(* Logix 5000 project; controller ARS14002_PLC vendor 1 type 14 code 218 rev 30.11; software revision 30.01; part 3 of 13 *)
(* tags used below, declared in another part *)
   AC_OK_1000 : BOOL;
   AC_OK_600 : BOOL;
   AC_OK_800 : BOOL;
   AC_OK_MCP : BOOL;
   AN_1000A : CM_AI_SCL;
   AN_1000B : CM_AI_SCL;
   AN_1000C : CM_AI_SCL;
   AN_101A : CM_AI_SCL;
   AN_101B : CM_AI_SCL;
   AN_101C : CM_AI_SCL;
   AN_200A : CM_AI_SCL;
   ARS_TO_AT3 : UDT_IPC;
   AT2_ATOMIZE_FLOW : REAL;
   AT2_ATOMIZE_FLOW_SCFM : REAL;
   AT2_CHAMBER_PRESSURE : REAL;
   AT2_COMM_STATUS_CONS : BOOL;
   AT2_COMM_STATUS_PROD : BOOL;
   AT2_END_ATOMIZATION : BOOL;
   AT2_HIBON_DISCHARGE_TEMP : REAL;
   AT2_HIBON_INSERTION_VALVE_OPEN : BOOL;
   AT2_HIBON_RUNNING : BOOL;
   AT2_INLET_FLOW : REAL;
   AT2_INLET_FLOW_SCFM : REAL;
   AT2_INLET_VALVE_OPEN : BOOL;
   AT2_PARTICULATE_POST_CYCLONE : REAL;
   AT2_PARTICULATE_POST_FILTER : REAL;
   AT2_PEDESTAL_LEVEL : REAL;
   AT2_PRAXAIR_PRESSURE : REAL;
   AT2_PRESTART : BOOL;
   AT2_START_ATOMIZATION : BOOL;
   AT2_V1_OPEN : BOOL;
   AT2_V4_OPEN : BOOL;
   AT3_ATOMIZE_FLOW : REAL;
   AT3_ATOMIZE_FLOW_SCFM : REAL;
   AT3_ATOMIZE_VALVE_OPEN : BOOL;
   AT3_CHAMBER_PRESSURE : REAL;
   AT3_CHAMBER_VACUUM : REAL;
   AT3_COMM_STATUS_CONS : BOOL;
   AT3_COMM_STATUS_PROD : BOOL;
   AT3_END_ATOMIZATION : BOOL;
   AT3_HIBON_DISCHARGE_TEMP : REAL;
   AT3_HIBON_INSERTION_VALVE_OPEN : BOOL;
   AT3_HIBON_RUNNING : BOOL;
   AT3_INLET_FLOW : REAL;
   AT3_INLET_FLOW_SCFM : REAL;
   AT3_INLET_VALVE_OPEN : BOOL;
   AT3_MELT_STATUS : BOOL;
   AT3_PARTICULATE_POST_CYCLONE : REAL;
   AT3_PARTICULATE_POST_FILTER : REAL;
   AT3_PEDESTAL_LEVEL : REAL;
   AT3_PRESTART : BOOL;
   AT3_START_ATOMIZATION : BOOL;
   AT3_TO_ARS : UDT_IPC;
   AT3_V1_OPEN : BOOL;
   AT3_V4_OPEN : BOOL;
   DC_OK_1000 : BOOL;
   DC_OK_600 : BOOL;
   DC_OK_800 : BOOL;
   DC_OK_MCP : BOOL;
   Deoxo_CurrentState : DINT;
   Deoxo_TransitionState : DINT;
   ESTOP_1 : BOOL;   // Pump Skid E-Stops
   ESTOP_2 : BOOL;   // FAN/HXR E-Stops
   ew_test_200 : BOOL;
   FSL_1000B : BOOL;
   FT_1002 : CM_AI_SCL;
   FT_1221 : CM_AI_SCL;
   FT_1251 : CM_AI_SCL;
   FT_202 : CM_AI_SCL;
   FT_202_ALT_SCFM : REAL;
   FT_502 : CM_AI_SCL;
   FT_502_ALT_SCFM : REAL;
   FT_904 : CM_AI_SCL;
   HXR_1250 : CM_DO_FVNR;
   IT_1250 : CM_AI_SCL;
   MTR_550 : CM_DO_FVNR;
   P_800A_RUN_OCCURRED : BOOL;
   P_800B_RUN_OCCURRED : BOOL;
   P_800C : CM_DO_FVR;
   P_800C_RUN_OCCURRED : BOOL;
   P_800D : CM_DO_FVR;
   P_800D_RUN_OCCURRED : BOOL;
   PDT_1101A : CM_AI_SCL_ALT;
   PDT_1301A : CM_AI_SCL_ALT;
   PDT_1301B : CM_AI_SCL_ALT;
   PDT_601 : CM_AI_SCL_ALT;
   PDT_603 : CM_AI_SCL_ALT;
   PDT_603_PERCENT : REAL;
   PDT_701 : CM_AI_SCL_ALT;
   PDT_701_ALT_GAL : REAL;
   PDT_701_ALT_SCF : REAL;
   PDT_721_CALC : REAL;
   PDT_751 : CM_AI_SCL_ALT;
   PDT_753 : CM_AI_SCL_ALT;
   PILOT_ATOMIZE_VALVE_OPEN : BOOL;   // Halo Valve
   PILOT_COMM_STATUS : BOOL;
   PILOT_EXHAUST_VALVE_OPEN : BOOL;
   PILOT_INLET_VALVE_OPEN : BOOL;   // Pressure Control Status (Backfill)
   PILOT_PARTICULATE_POST_FILTER : REAL;
   PILOT_PEDESTAL_LEVEL : REAL;
   PT_051 : CM_AI_SCL;
   PT_1001 : CM_AI_SCL;
   PT_1002 : CM_AI_SCL;
   PT_1003 : CM_AI_SCL;
   PT_101A : CM_AI_SCL;
   PT_101B : CM_AI_SCL;
   PT_101C : CM_AI_SCL;
   PT_1101A : CM_AI_SCL;
   PT_1201 : CM_AI_SCL;
   PT_1220 : CM_AI_SCL;
   PT_1222 : CM_AI_SCL;
   PT_1301A : CM_AI_SCL;
   PT_1301B : CM_AI_SCL;
   PT_201 : CM_AI_SCL;
   PT_222 : CM_AI_SCL;
   PT_601 : CM_AI_SCL;
   PT_601_LR : CM_AI_SCL;
   PT_603 : CM_AI_SCL;
   PT_701 : CM_AI_SCL;
   PT_721 : CM_AI_SCL;
   PT_751 : CM_AI_SCL;
   PT_753 : CM_AI_SCL;
   PT_802A : CM_AI_SCL;
   PT_802B : CM_AI_SCL;
   PT_802C : CM_AI_SCL;
   PT_802D : CM_AI_SCL;
   PT_803 : CM_AI_SCL;
   PT_806 : CM_AI_SCL;
   PT_902 : CM_AI_SCL;
   SCR_1250 : BOOL;   // HXR-1250 SCR Active Signal
   TE_1003 : CM_AI_SCL;
   TE_101A : CM_AI_SCL;
   TE_101B : CM_AI_SCL;
   TE_101C : CM_AI_SCL;
   TE_1201 : CM_AI_SCL;
   TE_1202 : CM_AI_SCL;
   TE_1203 : CM_AI_SCL;
   TE_1204 : CM_AI_SCL;
   TE_1205 : CM_AI_SCL;
   TE_1206 : CM_AI_SCL;
   TE_1250A : CM_AI_SCL;
   TE_1250B : CM_AI_SCL;
   TE_1252 : CM_AI_SCL;
   TE_501 : CM_AI_SCL;
   TE_504 : CM_AI_SCL;
   TE_601 : CM_AI_SCL;
   TE_602 : CM_AI_SCL;
   TE_604 : CM_AI_SCL;
   TE_609 : CM_AI_SCL;
   TE_801A : CM_AI_SCL;
   TE_801B : CM_AI_SCL;
   TE_801C : CM_AI_SCL;
   TE_801D : CM_AI_SCL;
   TE_802A : CM_AI_SCL;
   TE_802B : CM_AI_SCL;
   TE_802C : CM_AI_SCL;
   TE_802D : CM_AI_SCL;
   TE_803A : CM_AI_SCL;
   TE_803B : CM_AI_SCL;
   TE_803C : CM_AI_SCL;
   TE_803D : CM_AI_SCL;
   TE_804A : CM_AI_SCL;
   TE_804B : CM_AI_SCL;
   TE_804C : CM_AI_SCL;
   TE_804D : CM_AI_SCL;
   TE_901 : CM_AI_SCL;
   TE_902 : CM_AI_SCL;
   TE_903 : CM_AI_SCL;
   TE_904 : CM_AI_SCL;
   TE_T_RAWMAX : INT;
   TE_T_RAWMIN : INT;
   TK_1000_SCF : REAL;   // TOTAL SCF IN BUFFER
   VAPORIZER_WATER_DIFFERENTIAL : REAL;
   WATCHDOG_IN_100 : BOOL;
   WATCHDOG_IN_1000 : BOOL;
   WATCHDOG_IN_600 : BOOL;
   WATCHDOG_IN_800 : BOOL;
   XV_1001 : CM_DO_VLV;
   XV_101B : CM_DO_VLV;
   XV_101C : CM_DO_VLV;
   XV_1123 : CM_DO_VLV;
   XV_1201 : CM_DO_VLV;
   XV_1202 : CM_DO_VLV;
   XV_1203 : CM_DO_VLV;
   XV_1204 : CM_DO_VLV;
   XV_1205 : CM_DO_VLV;
   XV_623 : CM_DO_VLV;
   XV_703 : CM_DO_VLV;
   XV_721A : CM_DO_VLV;
   XV_721B : CM_DO_VLV;
   XV_801A : CM_DO_VLV;
   XV_801B : CM_DO_VLV;
   XV_801C : CM_DO_VLV;
   XV_801D : CM_DO_VLV;
   XV_806 : CM_DO_VLV;
   ZT_1001 : CM_AI_SCL;
   ZT_1002 : CM_AI_SCL;
   ZT_101A : CM_AI_SCL;
   ZT_101B : CM_AI_SCL;
   ZT_101C : CM_AI_SCL;
   ZT_102A : CM_AI_SCL;
   ZT_102B : CM_AI_SCL;
   ZT_102C : CM_AI_SCL;
   ZT_1221 : CM_AI_SCL;
   ZT_1251 : CM_AI_SCL;
   ZT_202 : CM_AI_SCL;
   ZT_204 : CM_AI_SCL;
   ZT_207 : CM_AI_SCL;
   ZT_504 : CM_AI_SCL;
   ZT_603 : CM_AI_SCL;
   ZT_605 : CM_AI_SCL;
   ZT_753 : CM_AI_SCL;
   ZT_754 : CM_AI_SCL;
   ZT_755 : CM_AI_SCL;
(* MainProgPeriodic, continued *)

ROUTINE MainRoutinePeriodic   (* ladder *)
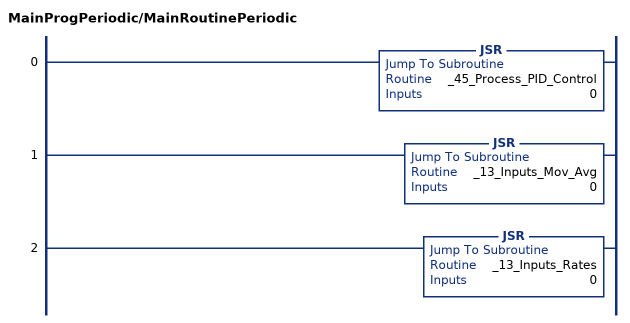
   0: JSR(_45_Process_PID_Control,0);
   1: JSR(_13_Inputs_Mov_Avg,0);
   2: JSR(_13_Inputs_Rates,0);
END_ROUTINE
END_PROGRAM

PROGRAM MainProgram   (* main routine MainRoutine *)
VAR
   BAND_01 : FBD_BOOLEAN_AND := (In3 := 1, In4 := 1, In5 := 1, In6 := 1, In7 := 1, In8 := 1);
   BNOT_01 : FBD_BOOLEAN_NOT := (Out := 1);
   BNOT_02 : FBD_BOOLEAN_NOT := (Out := 1);
   BNOT_03 : FBD_BOOLEAN_NOT := (Out := 1);
   BNOT_04 : FBD_BOOLEAN_NOT := (Out := 1);
   BOR_01 : FBD_BOOLEAN_OR;
   BOR_02 : FBD_BOOLEAN_OR;
   delete_ARS_DERIME_AUTO : BOOL;
   delete_AT2_PLANT_MAX_H2O : REAL := -85.0;
   delete_AT2_PLANT_MAX_O2 : REAL;
   delete_AT3_PLANT_MAX_H2O : REAL := -85.0;
   delete_AT3_PLANT_MAX_O2 : REAL;
   delete_PILOT_PLANT_MAX_H2O : REAL := -85.0;
   delete_PILOT_PLANT_MAX_O2 : REAL;
   delete_XV_623_FILL_MODE : BOOL;   // 0 = VENT 1 = FILL
   DERIME_EMPTY : BOOL;
   DERIME_EMPTY_ALARM : BOOL;
   DERIME_EMPTY_HOLD_TMR : TIMER := (PRE := 300000);
   DERIME_FILL : BOOL;
   DERIME_FULL : BOOL;
   DERIME_FULL_ALARM : BOOL;
   DERIME_FULL_HOLD_TMR : TIMER := (PRE := 600000);
   DERIME_SPH : REAL := 40.0;
   DERIME_SPL : REAL := 5.0;
   DERIME_VENT : BOOL := 1;
   DERV_01 : DERIVATIVE := (Gain := 1.0, RTSTime := 1);
   MAVE_01 : MOVING_AVERAGE := (SampleEnable := 1, NumberOfSamples := 1);
   MAVE_02 : MOVING_AVERAGE := (SampleEnable := 1, NumberOfSamples := 1);
   PT_701_DERIME_VENT_SPH : REAL := 30.0;
   PT_701_DERIME_VENT_SPL : REAL := 5.0;
   XV_721_BURP_TMR : TIMER;
END_VAR

ROUTINE _00_Startup   (* ladder *)
// Initialization Routines
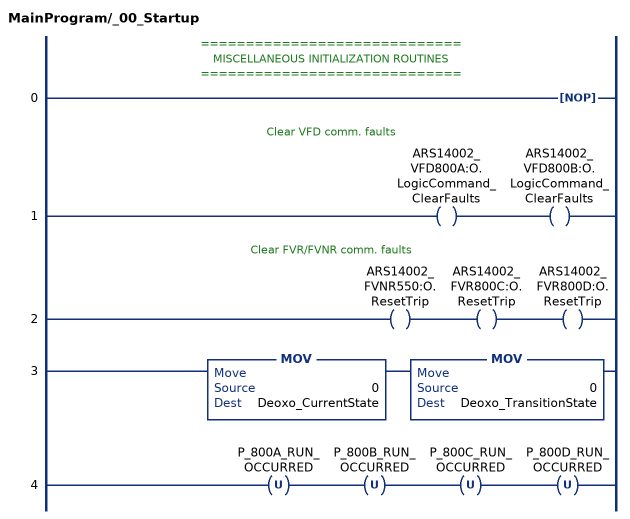
   // =============================
   // MISCELLANEOUS INITIALIZATION ROUTINES
   // =============================
   0: NOP();
   // Clear VFD comm. faults
   1: OTE(ARS14002_VFD800A:O.LogicCommand_ClearFaults)OTE(ARS14002_VFD800B:O.LogicCommand_ClearFaults);
   // Clear FVR/FVNR comm. faults
   2: OTE(ARS14002_FVNR550:O.ResetTrip)OTE(ARS14002_FVR800C:O.ResetTrip)OTE(ARS14002_FVR800D:O.ResetTrip);
   3: MOV(0,Deoxo_CurrentState)MOV(0,Deoxo_TransitionState);
   4: OTU(P_800A_RUN_OCCURRED)OTU(P_800B_RUN_OCCURRED)OTU(P_800C_RUN_OCCURRED)OTU(P_800D_RUN_OCCURRED);
END_ROUTINE

ROUTINE _10_Inputs_Analog   (* ladder *)
// Analog Input scaling and alarm handling routine
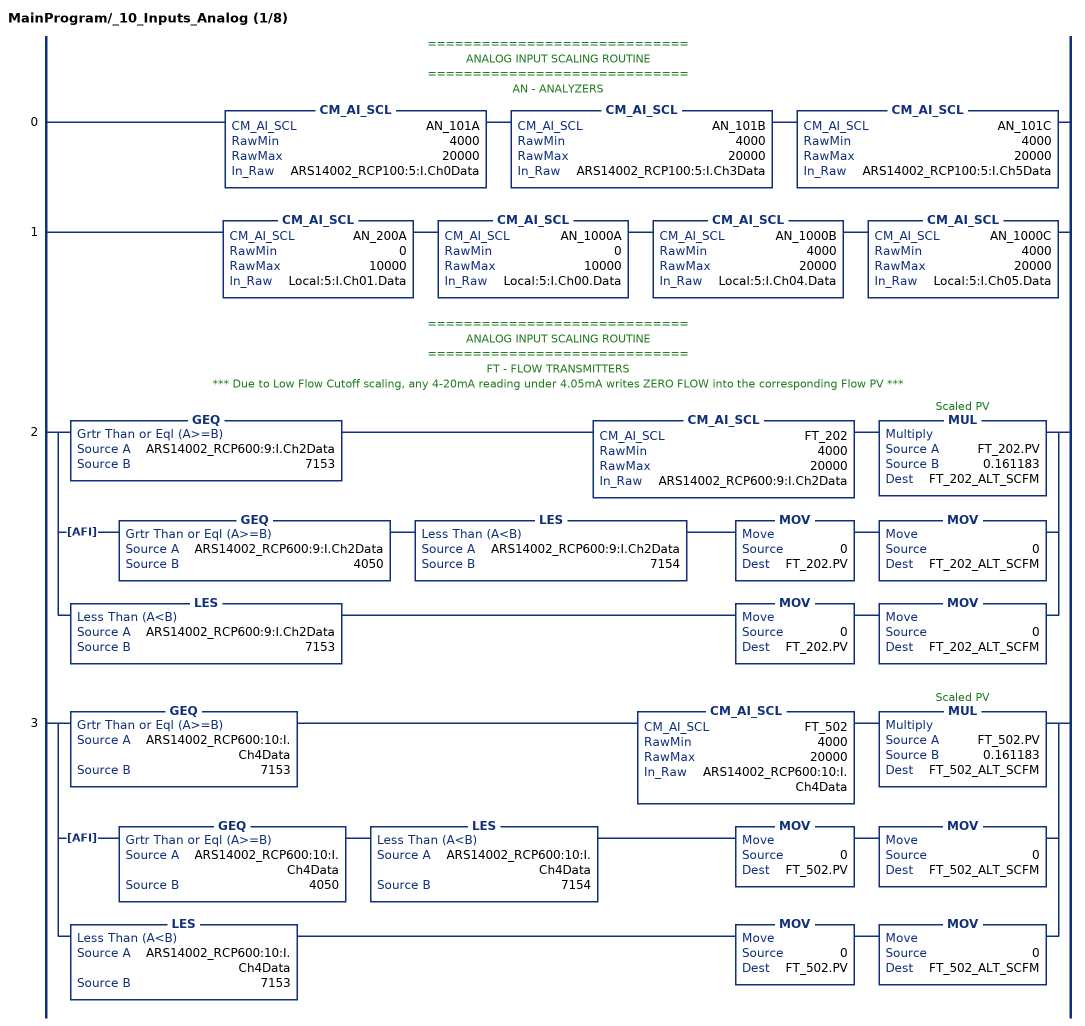
   // =============================
   // ANALOG INPUT SCALING ROUTINE
   // =============================
   // AN - ANALYZERS
   0: CM_AI_SCL(AN_101A,4000,20000,ARS14002_RCP100:5:I.Ch0Data)CM_AI_SCL(AN_101B,4000,20000,ARS14002_RCP100:5:I.Ch3Data)CM_AI_SCL(AN_101C,4000,20000,ARS14002_RCP100:5:I.Ch5Data);
   1: CM_AI_SCL(AN_200A,0,10000,Local:5:I.Ch01.Data)CM_AI_SCL(AN_1000A,0,10000,Local:5:I.Ch00.Data)CM_AI_SCL(AN_1000B,4000,20000,Local:5:I.Ch04.Data)CM_AI_SCL(AN_1000C,4000,20000,Local:5:I.Ch05.Data);
   // =============================
   // ANALOG INPUT SCALING ROUTINE
   // =============================
   // FT - FLOW TRANSMITTERS
   // *** Due to Low Flow Cutoff scaling, any 4-20mA reading under 4.05mA writes ZERO FLOW into the corresponding Flow PV ***
   2: [GEQ(ARS14002_RCP600:9:I.Ch2Data,7153) CM_AI_SCL(FT_202,4000,20000,ARS14002_RCP600:9:I.Ch2Data) MUL(FT_202.PV,0.161183,FT_202_ALT_SCFM) ,AFI() GEQ(ARS14002_RCP600:9:I.Ch2Data,4050) LES(ARS14002_RCP600:9:I.Ch2Data,7154) MOV(0,FT_202.PV) MOV(0,FT_202_ALT_SCFM) ,LES(ARS14002_RCP600:9:I.Ch2Data,7153) MOV(0,FT_202.PV) MOV(0,FT_202_ALT_SCFM) ];
   3: [GEQ(ARS14002_RCP600:10:I.Ch4Data,7153) CM_AI_SCL(FT_502,4000,20000,ARS14002_RCP600:10:I.Ch4Data) MUL(FT_502.PV,0.161183,FT_502_ALT_SCFM) ,AFI() GEQ(ARS14002_RCP600:10:I.Ch4Data,4050) LES(ARS14002_RCP600:10:I.Ch4Data,7154) MOV(0,FT_502.PV) MOV(0,FT_502_ALT_SCFM) ,LES(ARS14002_RCP600:10:I.Ch4Data,7153) MOV(0,FT_502.PV) MOV(0,FT_502_ALT_SCFM) ];
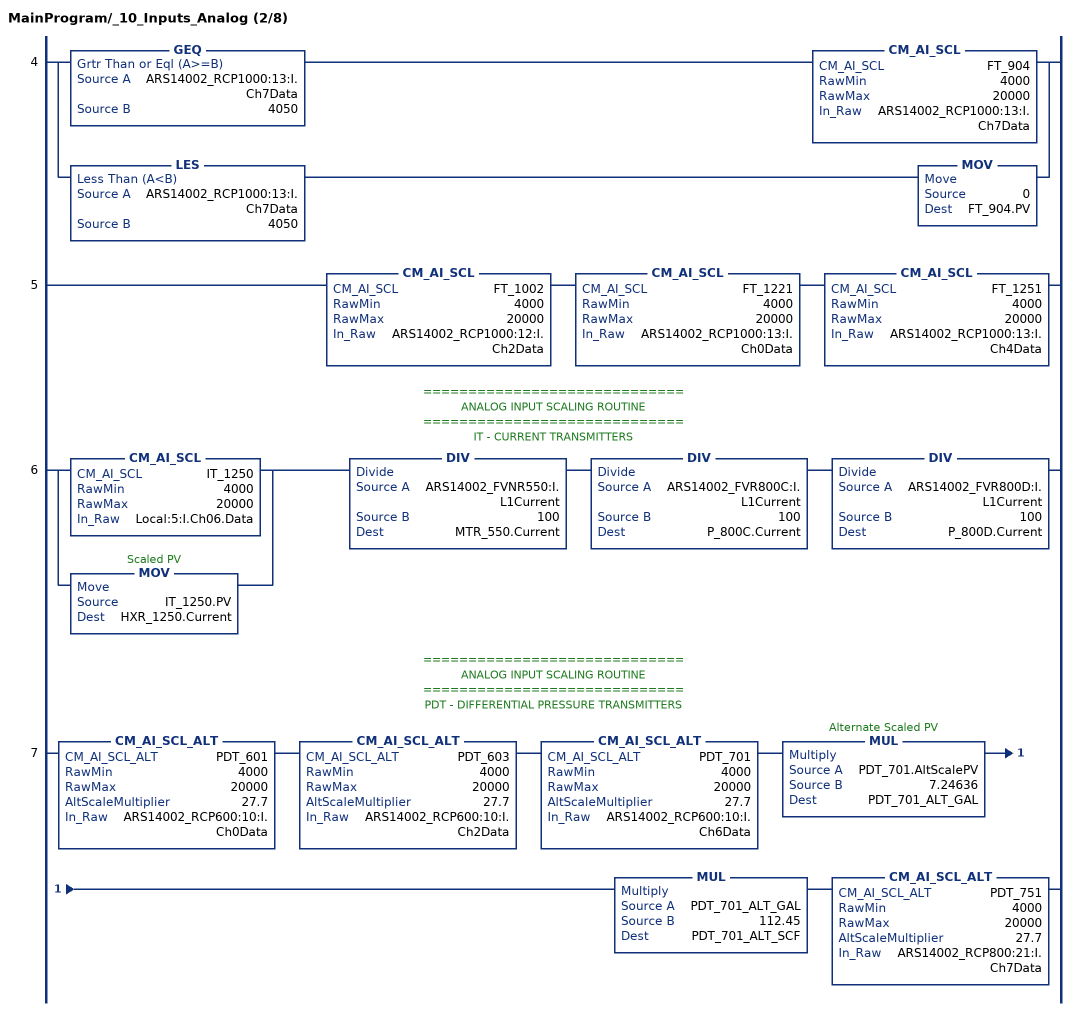
   4: [GEQ(ARS14002_RCP1000:13:I.Ch7Data,4050) CM_AI_SCL(FT_904,4000,20000,ARS14002_RCP1000:13:I.Ch7Data) ,LES(ARS14002_RCP1000:13:I.Ch7Data,4050) MOV(0,FT_904.PV) ];
   5: CM_AI_SCL(FT_1002,4000,20000,ARS14002_RCP1000:12:I.Ch2Data)CM_AI_SCL(FT_1221,4000,20000,ARS14002_RCP1000:13:I.Ch0Data)CM_AI_SCL(FT_1251,4000,20000,ARS14002_RCP1000:13:I.Ch4Data);
   // =============================
   // ANALOG INPUT SCALING ROUTINE
   // =============================
   // IT - CURRENT TRANSMITTERS
   6: [CM_AI_SCL(IT_1250,4000,20000,Local:5:I.Ch06.Data) ,MOV(IT_1250.PV,HXR_1250.Current) ]DIV(ARS14002_FVNR550:I.L1Current,100,MTR_550.Current)DIV(ARS14002_FVR800C:I.L1Current,100,P_800C.Current)DIV(ARS14002_FVR800D:I.L1Current,100,P_800D.Current);
   // =============================
   // ANALOG INPUT SCALING ROUTINE
   // =============================
   // PDT - DIFFERENTIAL PRESSURE TRANSMITTERS
   7: CM_AI_SCL_ALT(PDT_601,4000,20000,27.7,ARS14002_RCP600:10:I.Ch0Data)CM_AI_SCL_ALT(PDT_603,4000,20000,27.7,ARS14002_RCP600:10:I.Ch2Data)CM_AI_SCL_ALT(PDT_701,4000,20000,27.7,ARS14002_RCP600:10:I.Ch6Data)MUL(PDT_701.AltScalePV,7.24636,PDT_701_ALT_GAL)MUL(PDT_701_ALT_GAL,112.45,PDT_701_ALT_SCF)CM_AI_SCL_ALT(PDT_751,4000,20000,27.7,ARS14002_RCP800:21:I.Ch7Data);
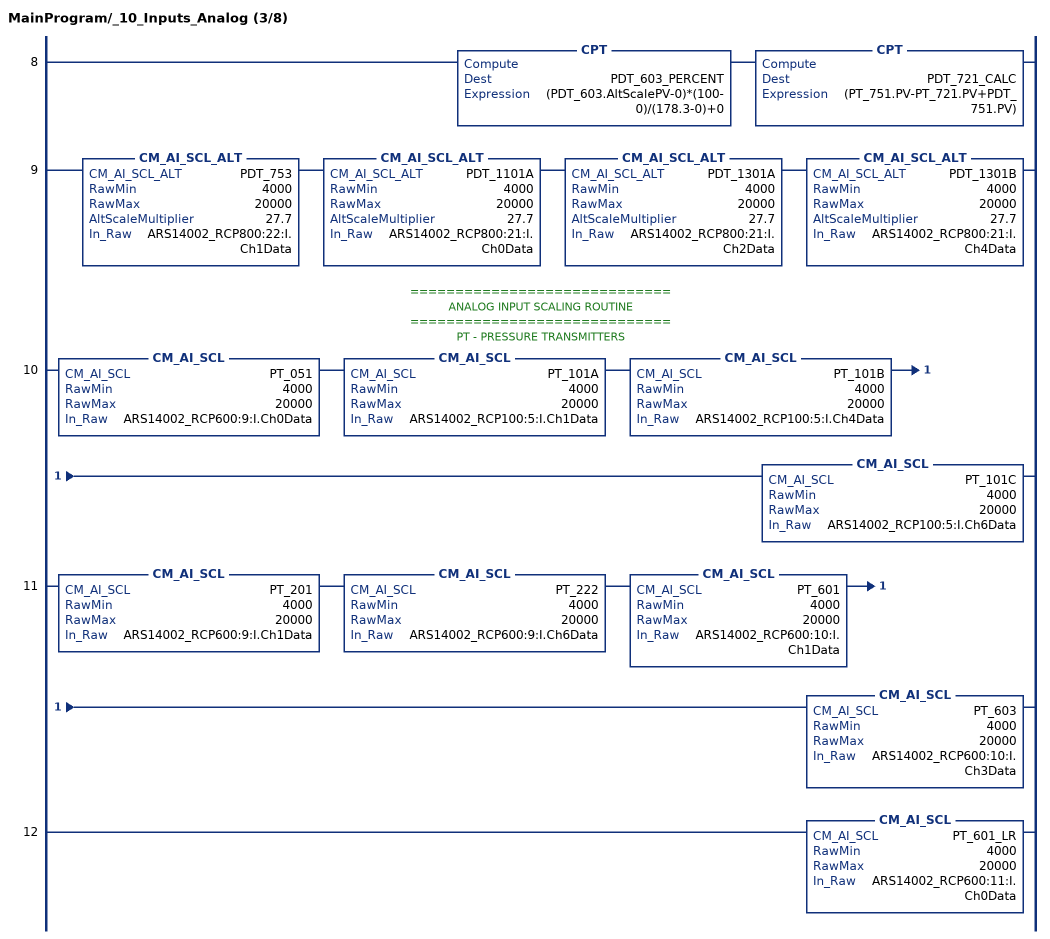
   8: CPT(PDT_603_PERCENT,(PDT_603.AltScalePV-0)*(100-0)/(178.3-0)+0)CPT(PDT_721_CALC,(PT_751.PV-PT_721.PV+PDT_751.PV));
   9: CM_AI_SCL_ALT(PDT_753,4000,20000,27.7,ARS14002_RCP800:22:I.Ch1Data)CM_AI_SCL_ALT(PDT_1101A,4000,20000,27.7,ARS14002_RCP800:21:I.Ch0Data)CM_AI_SCL_ALT(PDT_1301A,4000,20000,27.7,ARS14002_RCP800:21:I.Ch2Data)CM_AI_SCL_ALT(PDT_1301B,4000,20000,27.7,ARS14002_RCP800:21:I.Ch4Data);
   // =============================
   // ANALOG INPUT SCALING ROUTINE
   // =============================
   // PT - PRESSURE TRANSMITTERS
   10: CM_AI_SCL(PT_051,4000,20000,ARS14002_RCP600:9:I.Ch0Data)CM_AI_SCL(PT_101A,4000,20000,ARS14002_RCP100:5:I.Ch1Data)CM_AI_SCL(PT_101B,4000,20000,ARS14002_RCP100:5:I.Ch4Data)CM_AI_SCL(PT_101C,4000,20000,ARS14002_RCP100:5:I.Ch6Data);
   11: CM_AI_SCL(PT_201,4000,20000,ARS14002_RCP600:9:I.Ch1Data)CM_AI_SCL(PT_222,4000,20000,ARS14002_RCP600:9:I.Ch6Data)CM_AI_SCL(PT_601,4000,20000,ARS14002_RCP600:10:I.Ch1Data)CM_AI_SCL(PT_603,4000,20000,ARS14002_RCP600:10:I.Ch3Data);
   12: CM_AI_SCL(PT_601_LR,4000,20000,ARS14002_RCP600:11:I.Ch0Data);
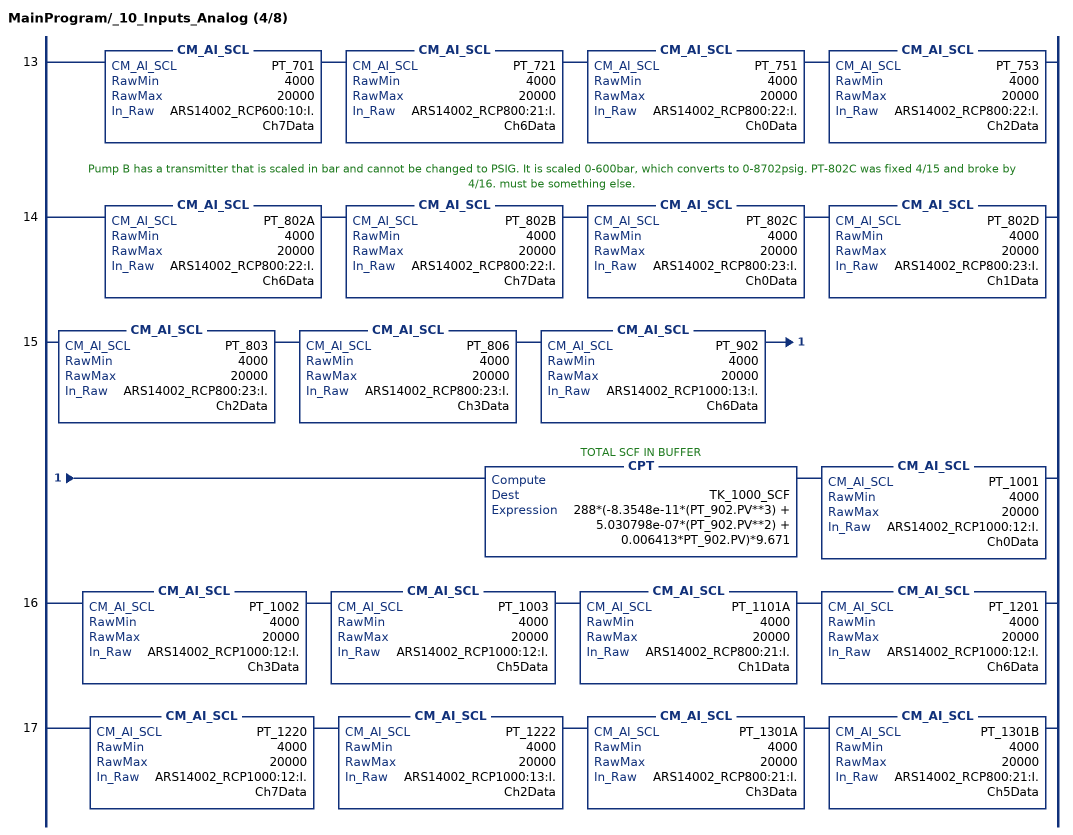
   13: CM_AI_SCL(PT_701,4000,20000,ARS14002_RCP600:10:I.Ch7Data)CM_AI_SCL(PT_721,4000,20000,ARS14002_RCP800:21:I.Ch6Data)CM_AI_SCL(PT_751,4000,20000,ARS14002_RCP800:22:I.Ch0Data)CM_AI_SCL(PT_753,4000,20000,ARS14002_RCP800:22:I.Ch2Data);
   // Pump B has a transmitter that is scaled in bar and cannot be changed to PSIG. It is scaled 0-600bar, which converts to 0-8702psig. PT-802C was fixed 4/15 and broke by 4/16. must be something else.
   14: CM_AI_SCL(PT_802A,4000,20000,ARS14002_RCP800:22:I.Ch6Data)CM_AI_SCL(PT_802B,4000,20000,ARS14002_RCP800:22:I.Ch7Data)CM_AI_SCL(PT_802C,4000,20000,ARS14002_RCP800:23:I.Ch0Data)CM_AI_SCL(PT_802D,4000,20000,ARS14002_RCP800:23:I.Ch1Data);
   15: CM_AI_SCL(PT_803,4000,20000,ARS14002_RCP800:23:I.Ch2Data)CM_AI_SCL(PT_806,4000,20000,ARS14002_RCP800:23:I.Ch3Data)CM_AI_SCL(PT_902,4000,20000,ARS14002_RCP1000:13:I.Ch6Data)CPT(TK_1000_SCF,288*(-8.3548e-11*(PT_902.PV**3) + 5.030798e-07*(PT_902.PV**2) + 0.006413*PT_902.PV)*9.671)CM_AI_SCL(PT_1001,4000,20000,ARS14002_RCP1000:12:I.Ch0Data);
   16: CM_AI_SCL(PT_1002,4000,20000,ARS14002_RCP1000:12:I.Ch3Data)CM_AI_SCL(PT_1003,4000,20000,ARS14002_RCP1000:12:I.Ch5Data)CM_AI_SCL(PT_1101A,4000,20000,ARS14002_RCP800:21:I.Ch1Data)CM_AI_SCL(PT_1201,4000,20000,ARS14002_RCP1000:12:I.Ch6Data);
   17: CM_AI_SCL(PT_1220,4000,20000,ARS14002_RCP1000:12:I.Ch7Data)CM_AI_SCL(PT_1222,4000,20000,ARS14002_RCP1000:13:I.Ch2Data)CM_AI_SCL(PT_1301A,4000,20000,ARS14002_RCP800:21:I.Ch3Data)CM_AI_SCL(PT_1301B,4000,20000,ARS14002_RCP800:21:I.Ch5Data);
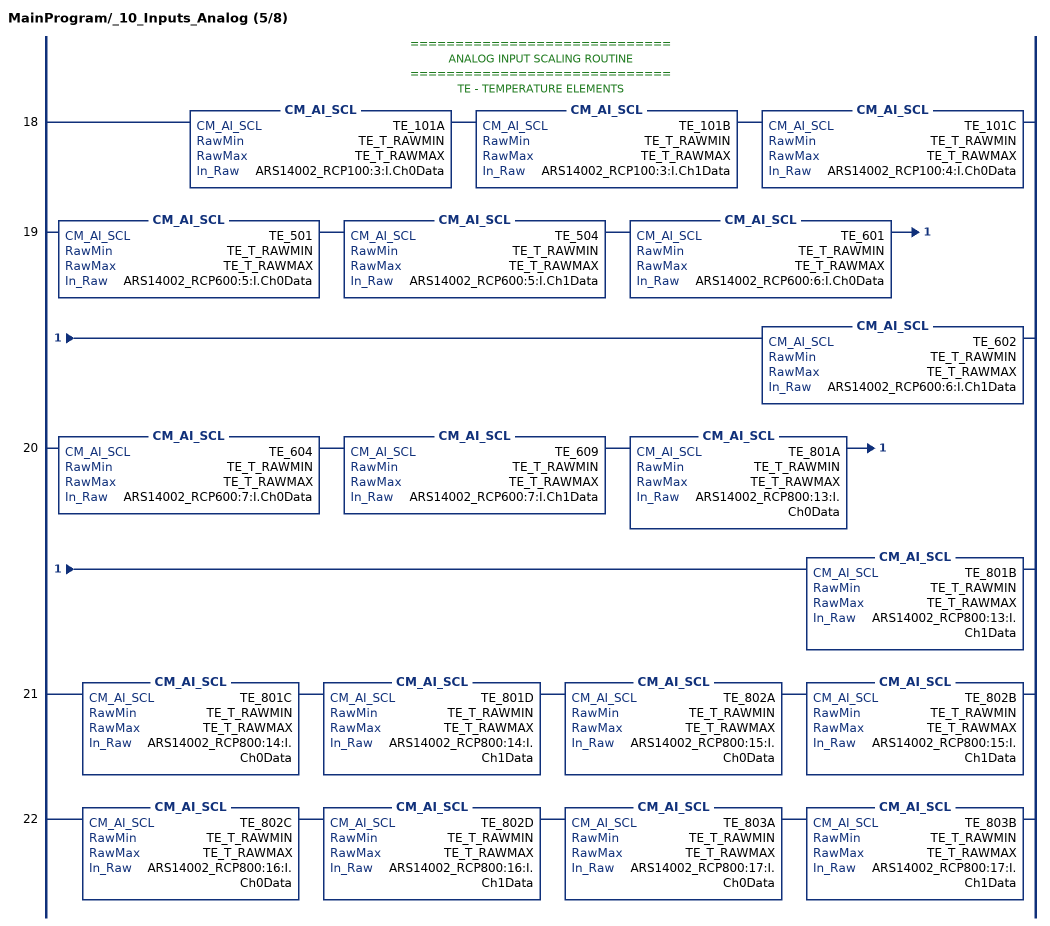
   // =============================
   // ANALOG INPUT SCALING ROUTINE
   // =============================
   // TE - TEMPERATURE ELEMENTS
   18: CM_AI_SCL(TE_101A,TE_T_RAWMIN,TE_T_RAWMAX,ARS14002_RCP100:3:I.Ch0Data)CM_AI_SCL(TE_101B,TE_T_RAWMIN,TE_T_RAWMAX,ARS14002_RCP100:3:I.Ch1Data)CM_AI_SCL(TE_101C,TE_T_RAWMIN,TE_T_RAWMAX,ARS14002_RCP100:4:I.Ch0Data);
   19: CM_AI_SCL(TE_501,TE_T_RAWMIN,TE_T_RAWMAX,ARS14002_RCP600:5:I.Ch0Data)CM_AI_SCL(TE_504,TE_T_RAWMIN,TE_T_RAWMAX,ARS14002_RCP600:5:I.Ch1Data)CM_AI_SCL(TE_601,TE_T_RAWMIN,TE_T_RAWMAX,ARS14002_RCP600:6:I.Ch0Data)CM_AI_SCL(TE_602,TE_T_RAWMIN,TE_T_RAWMAX,ARS14002_RCP600:6:I.Ch1Data);
   20: CM_AI_SCL(TE_604,TE_T_RAWMIN,TE_T_RAWMAX,ARS14002_RCP600:7:I.Ch0Data)CM_AI_SCL(TE_609,TE_T_RAWMIN,TE_T_RAWMAX,ARS14002_RCP600:7:I.Ch1Data)CM_AI_SCL(TE_801A,TE_T_RAWMIN,TE_T_RAWMAX,ARS14002_RCP800:13:I.Ch0Data)CM_AI_SCL(TE_801B,TE_T_RAWMIN,TE_T_RAWMAX,ARS14002_RCP800:13:I.Ch1Data);
   21: CM_AI_SCL(TE_801C,TE_T_RAWMIN,TE_T_RAWMAX,ARS14002_RCP800:14:I.Ch0Data)CM_AI_SCL(TE_801D,TE_T_RAWMIN,TE_T_RAWMAX,ARS14002_RCP800:14:I.Ch1Data)CM_AI_SCL(TE_802A,TE_T_RAWMIN,TE_T_RAWMAX,ARS14002_RCP800:15:I.Ch0Data)CM_AI_SCL(TE_802B,TE_T_RAWMIN,TE_T_RAWMAX,ARS14002_RCP800:15:I.Ch1Data);
   22: CM_AI_SCL(TE_802C,TE_T_RAWMIN,TE_T_RAWMAX,ARS14002_RCP800:16:I.Ch0Data)CM_AI_SCL(TE_802D,TE_T_RAWMIN,TE_T_RAWMAX,ARS14002_RCP800:16:I.Ch1Data)CM_AI_SCL(TE_803A,TE_T_RAWMIN,TE_T_RAWMAX,ARS14002_RCP800:17:I.Ch0Data)CM_AI_SCL(TE_803B,TE_T_RAWMIN,TE_T_RAWMAX,ARS14002_RCP800:17:I.Ch1Data);
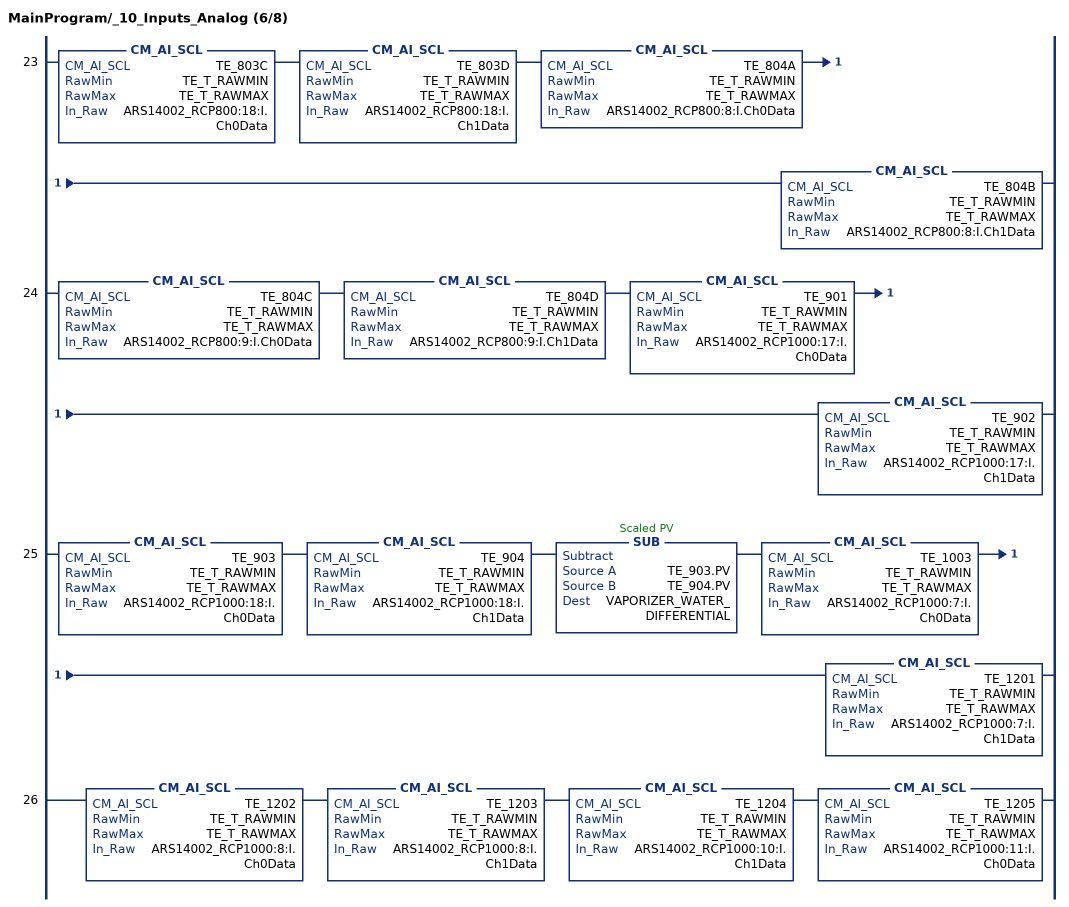
   23: CM_AI_SCL(TE_803C,TE_T_RAWMIN,TE_T_RAWMAX,ARS14002_RCP800:18:I.Ch0Data)CM_AI_SCL(TE_803D,TE_T_RAWMIN,TE_T_RAWMAX,ARS14002_RCP800:18:I.Ch1Data)CM_AI_SCL(TE_804A,TE_T_RAWMIN,TE_T_RAWMAX,ARS14002_RCP800:8:I.Ch0Data)CM_AI_SCL(TE_804B,TE_T_RAWMIN,TE_T_RAWMAX,ARS14002_RCP800:8:I.Ch1Data);
   24: CM_AI_SCL(TE_804C,TE_T_RAWMIN,TE_T_RAWMAX,ARS14002_RCP800:9:I.Ch0Data)CM_AI_SCL(TE_804D,TE_T_RAWMIN,TE_T_RAWMAX,ARS14002_RCP800:9:I.Ch1Data)CM_AI_SCL(TE_901,TE_T_RAWMIN,TE_T_RAWMAX,ARS14002_RCP1000:17:I.Ch0Data)CM_AI_SCL(TE_902,TE_T_RAWMIN,TE_T_RAWMAX,ARS14002_RCP1000:17:I.Ch1Data);
   25: CM_AI_SCL(TE_903,TE_T_RAWMIN,TE_T_RAWMAX,ARS14002_RCP1000:18:I.Ch0Data)CM_AI_SCL(TE_904,TE_T_RAWMIN,TE_T_RAWMAX,ARS14002_RCP1000:18:I.Ch1Data)SUB(TE_903.PV,TE_904.PV,VAPORIZER_WATER_DIFFERENTIAL)CM_AI_SCL(TE_1003,TE_T_RAWMIN,TE_T_RAWMAX,ARS14002_RCP1000:7:I.Ch0Data)CM_AI_SCL(TE_1201,TE_T_RAWMIN,TE_T_RAWMAX,ARS14002_RCP1000:7:I.Ch1Data);
   26: CM_AI_SCL(TE_1202,TE_T_RAWMIN,TE_T_RAWMAX,ARS14002_RCP1000:8:I.Ch0Data)CM_AI_SCL(TE_1203,TE_T_RAWMIN,TE_T_RAWMAX,ARS14002_RCP1000:8:I.Ch1Data)CM_AI_SCL(TE_1204,TE_T_RAWMIN,TE_T_RAWMAX,ARS14002_RCP1000:10:I.Ch1Data)CM_AI_SCL(TE_1205,TE_T_RAWMIN,TE_T_RAWMAX,ARS14002_RCP1000:11:I.Ch0Data);
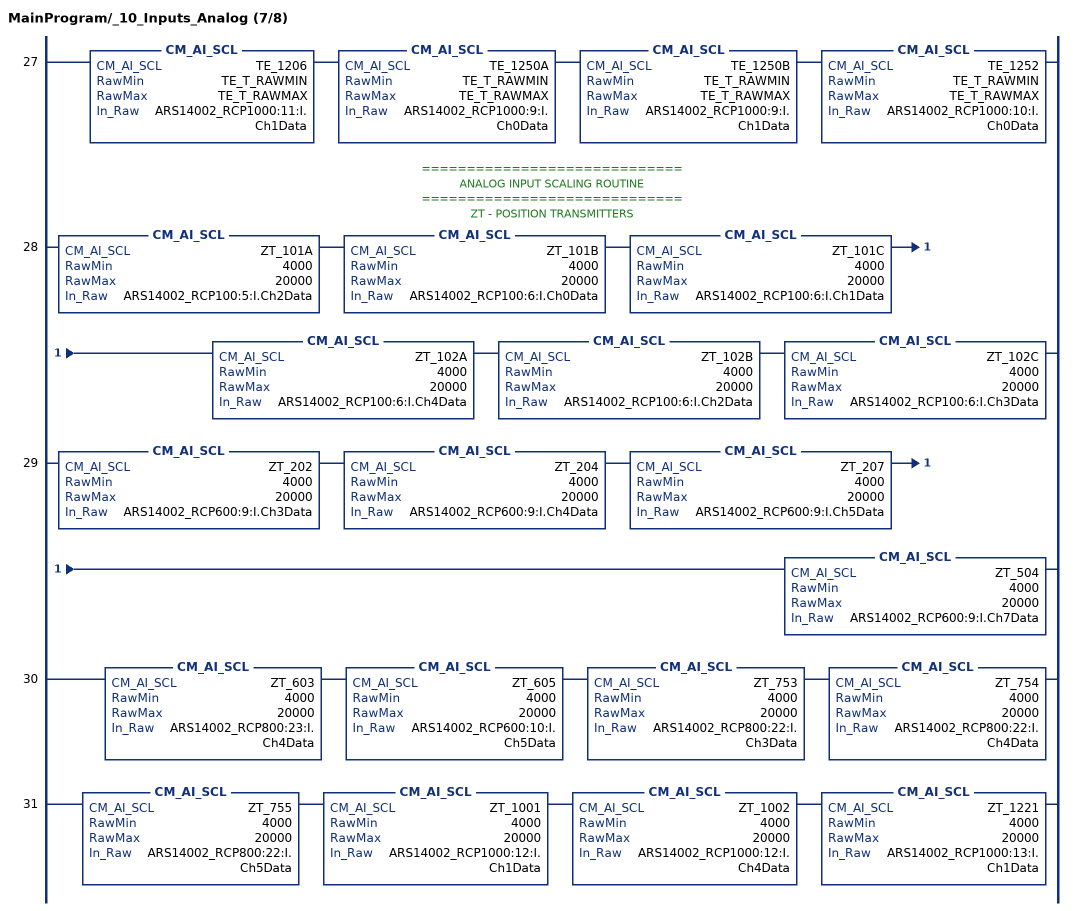
   27: CM_AI_SCL(TE_1206,TE_T_RAWMIN,TE_T_RAWMAX,ARS14002_RCP1000:11:I.Ch1Data)CM_AI_SCL(TE_1250A,TE_T_RAWMIN,TE_T_RAWMAX,ARS14002_RCP1000:9:I.Ch0Data)CM_AI_SCL(TE_1250B,TE_T_RAWMIN,TE_T_RAWMAX,ARS14002_RCP1000:9:I.Ch1Data)CM_AI_SCL(TE_1252,TE_T_RAWMIN,TE_T_RAWMAX,ARS14002_RCP1000:10:I.Ch0Data);
   // =============================
   // ANALOG INPUT SCALING ROUTINE
   // =============================
   // ZT - POSITION TRANSMITTERS
   28: CM_AI_SCL(ZT_101A,4000,20000,ARS14002_RCP100:5:I.Ch2Data)CM_AI_SCL(ZT_101B,4000,20000,ARS14002_RCP100:6:I.Ch0Data)CM_AI_SCL(ZT_101C,4000,20000,ARS14002_RCP100:6:I.Ch1Data)CM_AI_SCL(ZT_102A,4000,20000,ARS14002_RCP100:6:I.Ch4Data)CM_AI_SCL(ZT_102B,4000,20000,ARS14002_RCP100:6:I.Ch2Data)CM_AI_SCL(ZT_102C,4000,20000,ARS14002_RCP100:6:I.Ch3Data);
   29: CM_AI_SCL(ZT_202,4000,20000,ARS14002_RCP600:9:I.Ch3Data)CM_AI_SCL(ZT_204,4000,20000,ARS14002_RCP600:9:I.Ch4Data)CM_AI_SCL(ZT_207,4000,20000,ARS14002_RCP600:9:I.Ch5Data)CM_AI_SCL(ZT_504,4000,20000,ARS14002_RCP600:9:I.Ch7Data);
   30: CM_AI_SCL(ZT_603,4000,20000,ARS14002_RCP800:23:I.Ch4Data)CM_AI_SCL(ZT_605,4000,20000,ARS14002_RCP600:10:I.Ch5Data)CM_AI_SCL(ZT_753,4000,20000,ARS14002_RCP800:22:I.Ch3Data)CM_AI_SCL(ZT_754,4000,20000,ARS14002_RCP800:22:I.Ch4Data);
   31: CM_AI_SCL(ZT_755,4000,20000,ARS14002_RCP800:22:I.Ch5Data)CM_AI_SCL(ZT_1001,4000,20000,ARS14002_RCP1000:12:I.Ch1Data)CM_AI_SCL(ZT_1002,4000,20000,ARS14002_RCP1000:12:I.Ch4Data)CM_AI_SCL(ZT_1221,4000,20000,ARS14002_RCP1000:13:I.Ch1Data);
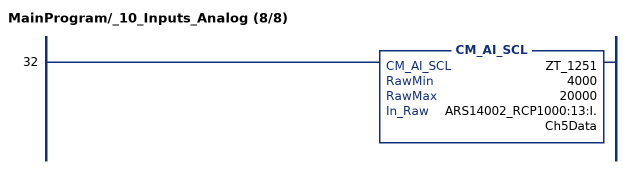
   32: CM_AI_SCL(ZT_1251,4000,20000,ARS14002_RCP1000:13:I.Ch5Data);
END_ROUTINE

ROUTINE _11_Inputs_Discrete   (* ladder *)
// Input Mapping Routine
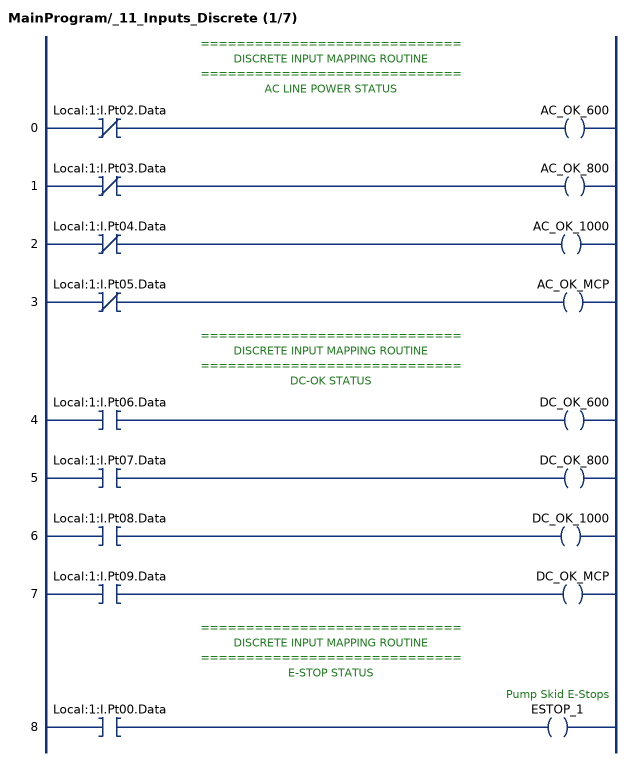
   // =============================
   // DISCRETE INPUT MAPPING ROUTINE
   // =============================
   // AC LINE POWER STATUS
   0: XIO(Local:1:I.Pt02.Data)OTE(AC_OK_600);
   1: XIO(Local:1:I.Pt03.Data)OTE(AC_OK_800);
   2: XIO(Local:1:I.Pt04.Data)OTE(AC_OK_1000);
   3: XIO(Local:1:I.Pt05.Data)OTE(AC_OK_MCP);
   // =============================
   // DISCRETE INPUT MAPPING ROUTINE
   // =============================
   // DC-OK STATUS
   4: XIC(Local:1:I.Pt06.Data)OTE(DC_OK_600);
   5: XIC(Local:1:I.Pt07.Data)OTE(DC_OK_800);
   6: XIC(Local:1:I.Pt08.Data)OTE(DC_OK_1000);
   7: XIC(Local:1:I.Pt09.Data)OTE(DC_OK_MCP);
   // =============================
   // DISCRETE INPUT MAPPING ROUTINE
   // =============================
   // E-STOP STATUS
   8: XIC(Local:1:I.Pt00.Data)OTE(ESTOP_1);
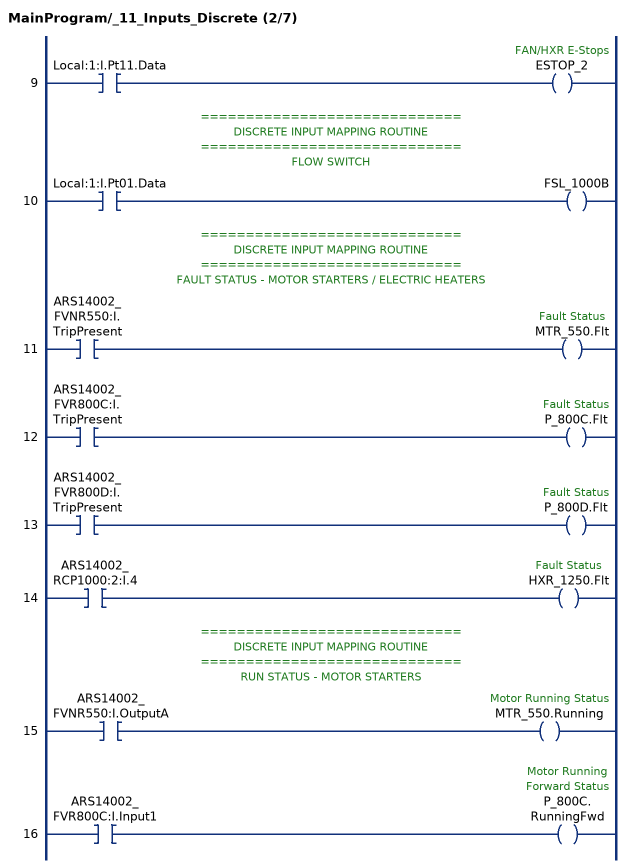
   9: XIC(Local:1:I.Pt11.Data)OTE(ESTOP_2);
   // =============================
   // DISCRETE INPUT MAPPING ROUTINE
   // =============================
   // FLOW SWITCH
   10: XIC(Local:1:I.Pt01.Data)OTE(FSL_1000B);
   // =============================
   // DISCRETE INPUT MAPPING ROUTINE
   // =============================
   // FAULT STATUS - MOTOR STARTERS / ELECTRIC HEATERS
   11: XIC(ARS14002_FVNR550:I.TripPresent)OTE(MTR_550.Flt);
   12: XIC(ARS14002_FVR800C:I.TripPresent)OTE(P_800C.Flt);
   13: XIC(ARS14002_FVR800D:I.TripPresent)OTE(P_800D.Flt);
   14: XIC(ARS14002_RCP1000:2:I.4)OTE(HXR_1250.Flt);
   // =============================
   // DISCRETE INPUT MAPPING ROUTINE
   // =============================
   // RUN STATUS - MOTOR STARTERS
   15: XIC(ARS14002_FVNR550:I.OutputA)OTE(MTR_550.Running);
   16: XIC(ARS14002_FVR800C:I.Input1)OTE(P_800C.RunningFwd);
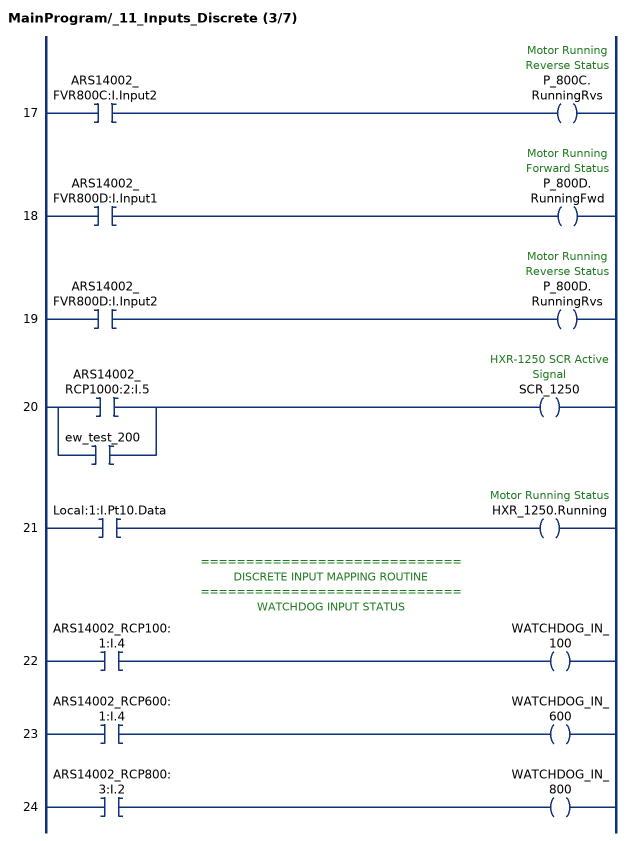
   17: XIC(ARS14002_FVR800C:I.Input2)OTE(P_800C.RunningRvs);
   18: XIC(ARS14002_FVR800D:I.Input1)OTE(P_800D.RunningFwd);
   19: XIC(ARS14002_FVR800D:I.Input2)OTE(P_800D.RunningRvs);
   20: [XIC(ARS14002_RCP1000:2:I.5) ,XIC(ew_test_200) ]OTE(SCR_1250);
   21: XIC(Local:1:I.Pt10.Data)OTE(HXR_1250.Running);
   // =============================
   // DISCRETE INPUT MAPPING ROUTINE
   // =============================
   // WATCHDOG INPUT STATUS
   22: XIC(ARS14002_RCP100:1:I.4)OTE(WATCHDOG_IN_100);
   23: XIC(ARS14002_RCP600:1:I.4)OTE(WATCHDOG_IN_600);
   24: XIC(ARS14002_RCP800:3:I.2)OTE(WATCHDOG_IN_800);
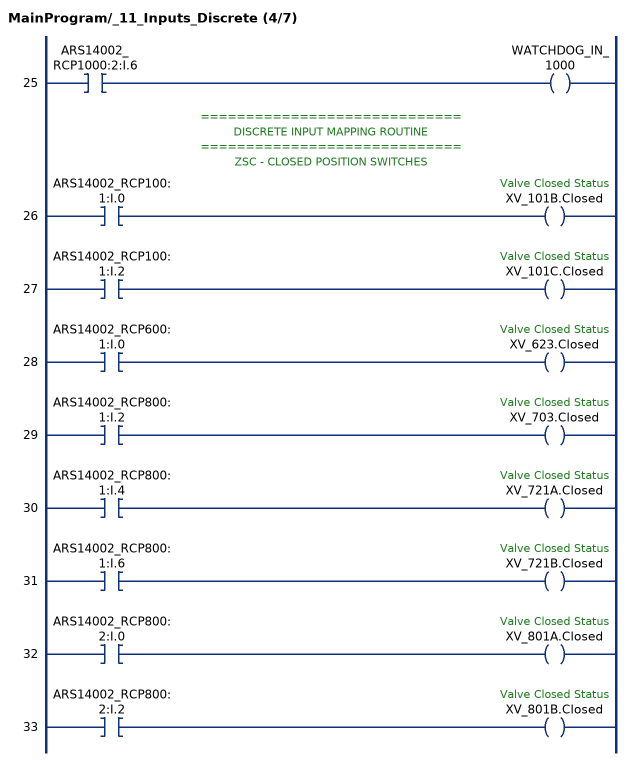
   25: XIC(ARS14002_RCP1000:2:I.6)OTE(WATCHDOG_IN_1000);
   // =============================
   // DISCRETE INPUT MAPPING ROUTINE
   // =============================
   // ZSC - CLOSED POSITION SWITCHES
   26: XIC(ARS14002_RCP100:1:I.0)OTE(XV_101B.Closed);
   27: XIC(ARS14002_RCP100:1:I.2)OTE(XV_101C.Closed);
   28: XIC(ARS14002_RCP600:1:I.0)OTE(XV_623.Closed);
   29: XIC(ARS14002_RCP800:1:I.2)OTE(XV_703.Closed);
   30: XIC(ARS14002_RCP800:1:I.4)OTE(XV_721A.Closed);
   31: XIC(ARS14002_RCP800:1:I.6)OTE(XV_721B.Closed);
   32: XIC(ARS14002_RCP800:2:I.0)OTE(XV_801A.Closed);
   33: XIC(ARS14002_RCP800:2:I.2)OTE(XV_801B.Closed);
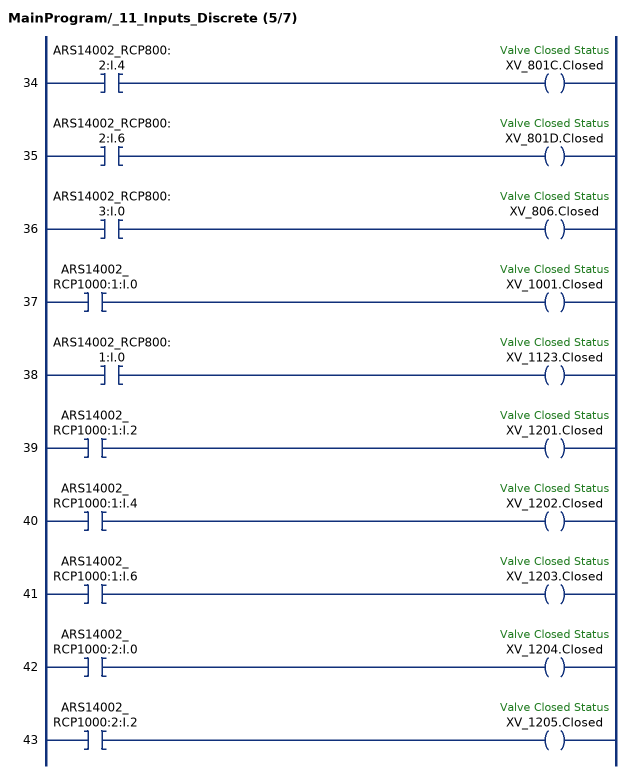
   34: XIC(ARS14002_RCP800:2:I.4)OTE(XV_801C.Closed);
   35: XIC(ARS14002_RCP800:2:I.6)OTE(XV_801D.Closed);
   36: XIC(ARS14002_RCP800:3:I.0)OTE(XV_806.Closed);
   37: XIC(ARS14002_RCP1000:1:I.0)OTE(XV_1001.Closed);
   38: XIC(ARS14002_RCP800:1:I.0)OTE(XV_1123.Closed);
   39: XIC(ARS14002_RCP1000:1:I.2)OTE(XV_1201.Closed);
   40: XIC(ARS14002_RCP1000:1:I.4)OTE(XV_1202.Closed);
   41: XIC(ARS14002_RCP1000:1:I.6)OTE(XV_1203.Closed);
   42: XIC(ARS14002_RCP1000:2:I.0)OTE(XV_1204.Closed);
   43: XIC(ARS14002_RCP1000:2:I.2)OTE(XV_1205.Closed);
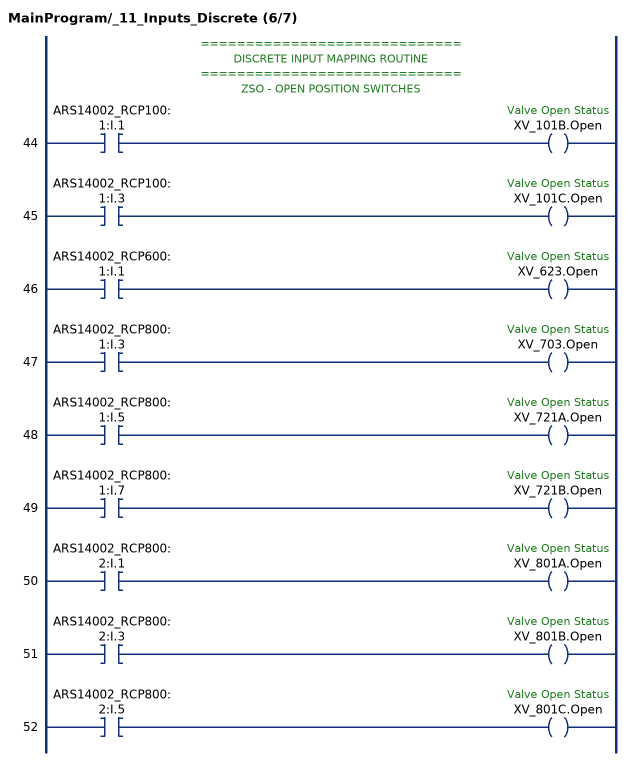
   // =============================
   // DISCRETE INPUT MAPPING ROUTINE
   // =============================
   // ZSO - OPEN POSITION SWITCHES
   44: XIC(ARS14002_RCP100:1:I.1)OTE(XV_101B.Open);
   45: XIC(ARS14002_RCP100:1:I.3)OTE(XV_101C.Open);
   46: XIC(ARS14002_RCP600:1:I.1)OTE(XV_623.Open);
   47: XIC(ARS14002_RCP800:1:I.3)OTE(XV_703.Open);
   48: XIC(ARS14002_RCP800:1:I.5)OTE(XV_721A.Open);
   49: XIC(ARS14002_RCP800:1:I.7)OTE(XV_721B.Open);
   50: XIC(ARS14002_RCP800:2:I.1)OTE(XV_801A.Open);
   51: XIC(ARS14002_RCP800:2:I.3)OTE(XV_801B.Open);
   52: XIC(ARS14002_RCP800:2:I.5)OTE(XV_801C.Open);
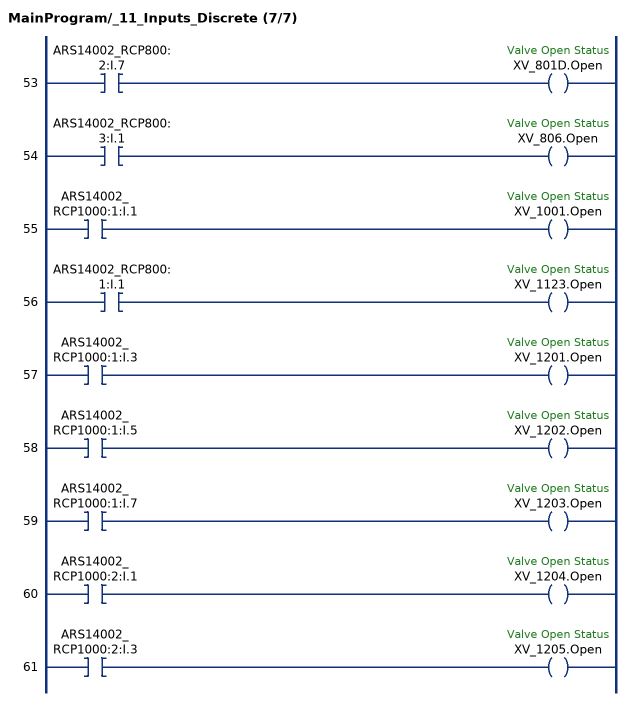
   53: XIC(ARS14002_RCP800:2:I.7)OTE(XV_801D.Open);
   54: XIC(ARS14002_RCP800:3:I.1)OTE(XV_806.Open);
   55: XIC(ARS14002_RCP1000:1:I.1)OTE(XV_1001.Open);
   56: XIC(ARS14002_RCP800:1:I.1)OTE(XV_1123.Open);
   57: XIC(ARS14002_RCP1000:1:I.3)OTE(XV_1201.Open);
   58: XIC(ARS14002_RCP1000:1:I.5)OTE(XV_1202.Open);
   59: XIC(ARS14002_RCP1000:1:I.7)OTE(XV_1203.Open);
   60: XIC(ARS14002_RCP1000:2:I.1)OTE(XV_1204.Open);
   61: XIC(ARS14002_RCP1000:2:I.3)OTE(XV_1205.Open);
END_ROUTINE

ROUTINE _12_Inputs_IPC   (* ladder *)
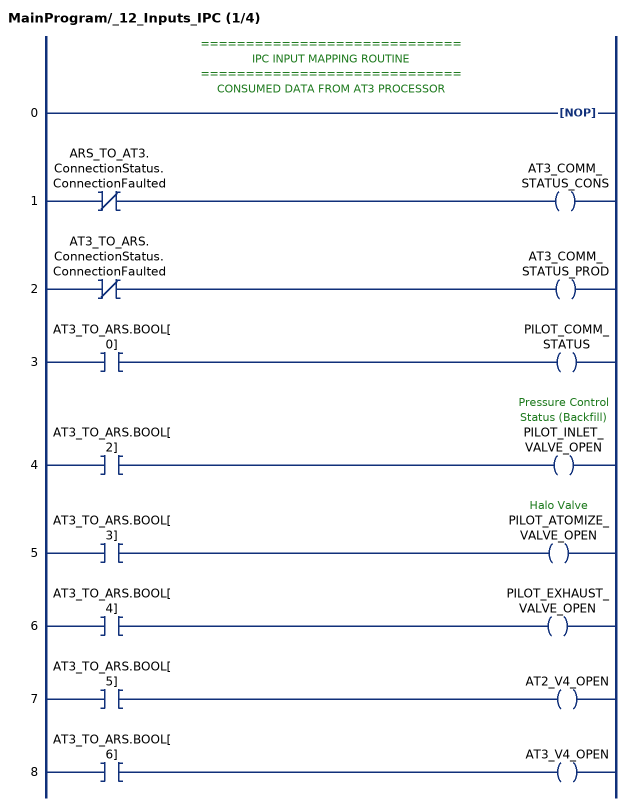
   // =============================
   // IPC INPUT MAPPING ROUTINE
   // =============================
   // CONSUMED DATA FROM AT3 PROCESSOR
   0: NOP();
   1: XIO(ARS_TO_AT3.ConnectionStatus.ConnectionFaulted)OTE(AT3_COMM_STATUS_CONS);
   2: XIO(AT3_TO_ARS.ConnectionStatus.ConnectionFaulted)OTE(AT3_COMM_STATUS_PROD);
   3: XIC(AT3_TO_ARS.BOOL[0])OTE(PILOT_COMM_STATUS);
   4: XIC(AT3_TO_ARS.BOOL[2])OTE(PILOT_INLET_VALVE_OPEN);
   5: XIC(AT3_TO_ARS.BOOL[3])OTE(PILOT_ATOMIZE_VALVE_OPEN);
   6: XIC(AT3_TO_ARS.BOOL[4])OTE(PILOT_EXHAUST_VALVE_OPEN);
   7: XIC(AT3_TO_ARS.BOOL[5])OTE(AT2_V4_OPEN);
   8: XIC(AT3_TO_ARS.BOOL[6])OTE(AT3_V4_OPEN);
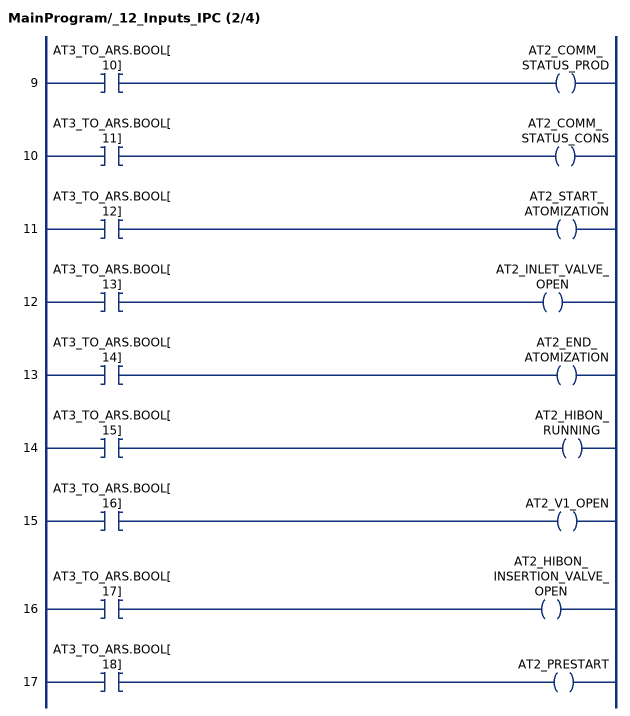
   9: XIC(AT3_TO_ARS.BOOL[10])OTE(AT2_COMM_STATUS_PROD);
   10: XIC(AT3_TO_ARS.BOOL[11])OTE(AT2_COMM_STATUS_CONS);
   11: XIC(AT3_TO_ARS.BOOL[12])OTE(AT2_START_ATOMIZATION);
   12: XIC(AT3_TO_ARS.BOOL[13])OTE(AT2_INLET_VALVE_OPEN);
   13: XIC(AT3_TO_ARS.BOOL[14])OTE(AT2_END_ATOMIZATION);
   14: XIC(AT3_TO_ARS.BOOL[15])OTE(AT2_HIBON_RUNNING);
   15: XIC(AT3_TO_ARS.BOOL[16])OTE(AT2_V1_OPEN);
   16: XIC(AT3_TO_ARS.BOOL[17])OTE(AT2_HIBON_INSERTION_VALVE_OPEN);
   17: XIC(AT3_TO_ARS.BOOL[18])OTE(AT2_PRESTART);
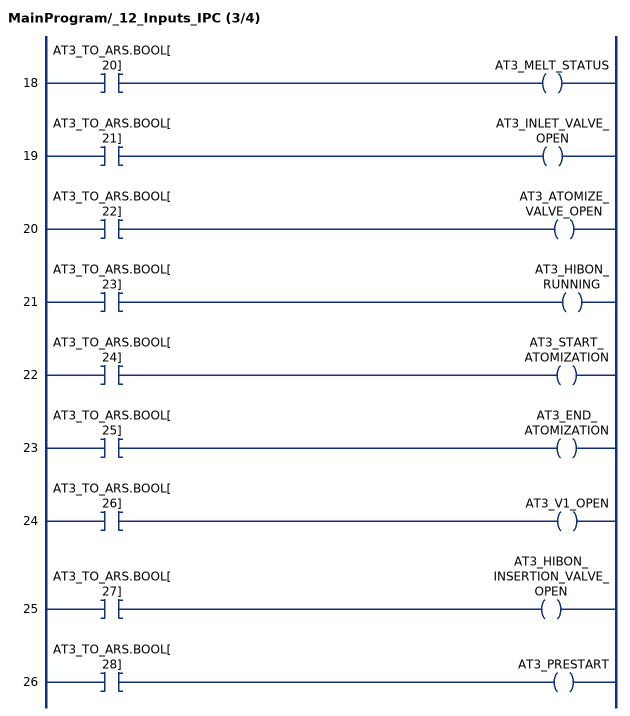
   18: XIC(AT3_TO_ARS.BOOL[20])OTE(AT3_MELT_STATUS);
   19: XIC(AT3_TO_ARS.BOOL[21])OTE(AT3_INLET_VALVE_OPEN);
   20: XIC(AT3_TO_ARS.BOOL[22])OTE(AT3_ATOMIZE_VALVE_OPEN);
   21: XIC(AT3_TO_ARS.BOOL[23])OTE(AT3_HIBON_RUNNING);
   22: XIC(AT3_TO_ARS.BOOL[24])OTE(AT3_START_ATOMIZATION);
   23: XIC(AT3_TO_ARS.BOOL[25])OTE(AT3_END_ATOMIZATION);
   24: XIC(AT3_TO_ARS.BOOL[26])OTE(AT3_V1_OPEN);
   25: XIC(AT3_TO_ARS.BOOL[27])OTE(AT3_HIBON_INSERTION_VALVE_OPEN);
   26: XIC(AT3_TO_ARS.BOOL[28])OTE(AT3_PRESTART);
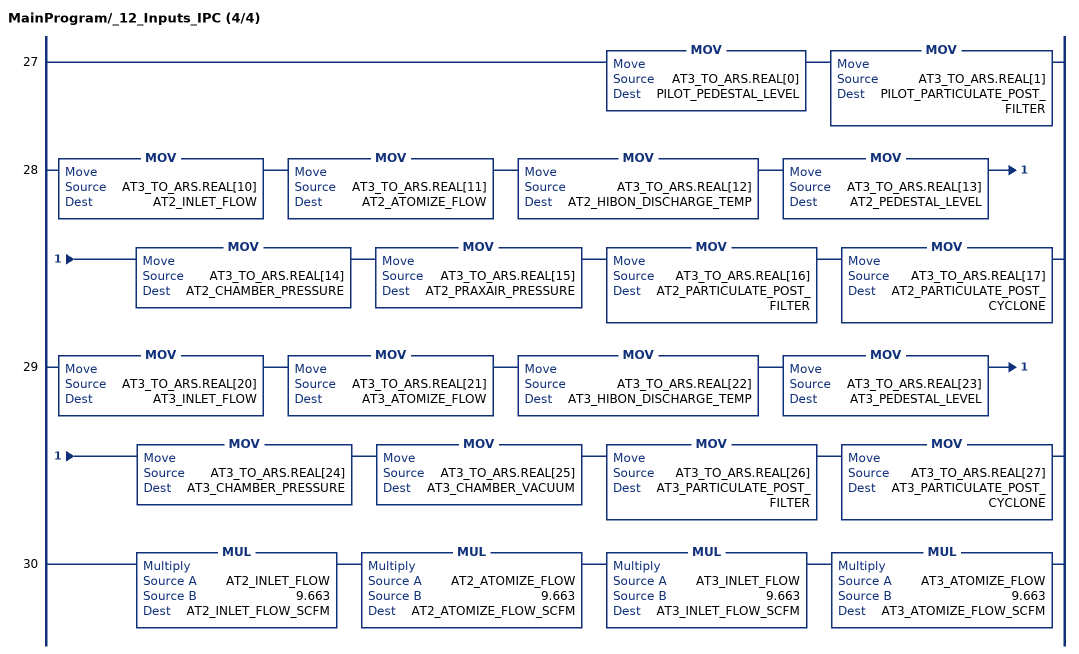
   27: MOV(AT3_TO_ARS.REAL[0],PILOT_PEDESTAL_LEVEL)MOV(AT3_TO_ARS.REAL[1],PILOT_PARTICULATE_POST_FILTER);
   28: MOV(AT3_TO_ARS.REAL[10],AT2_INLET_FLOW)MOV(AT3_TO_ARS.REAL[11],AT2_ATOMIZE_FLOW)MOV(AT3_TO_ARS.REAL[12],AT2_HIBON_DISCHARGE_TEMP)MOV(AT3_TO_ARS.REAL[13],AT2_PEDESTAL_LEVEL)MOV(AT3_TO_ARS.REAL[14],AT2_CHAMBER_PRESSURE)MOV(AT3_TO_ARS.REAL[15],AT2_PRAXAIR_PRESSURE)MOV(AT3_TO_ARS.REAL[16],AT2_PARTICULATE_POST_FILTER)MOV(AT3_TO_ARS.REAL[17],AT2_PARTICULATE_POST_CYCLONE);
   29: MOV(AT3_TO_ARS.REAL[20],AT3_INLET_FLOW)MOV(AT3_TO_ARS.REAL[21],AT3_ATOMIZE_FLOW)MOV(AT3_TO_ARS.REAL[22],AT3_HIBON_DISCHARGE_TEMP)MOV(AT3_TO_ARS.REAL[23],AT3_PEDESTAL_LEVEL)MOV(AT3_TO_ARS.REAL[24],AT3_CHAMBER_PRESSURE)MOV(AT3_TO_ARS.REAL[25],AT3_CHAMBER_VACUUM)MOV(AT3_TO_ARS.REAL[26],AT3_PARTICULATE_POST_FILTER)MOV(AT3_TO_ARS.REAL[27],AT3_PARTICULATE_POST_CYCLONE);
   30: MUL(AT2_INLET_FLOW,9.663,AT2_INLET_FLOW_SCFM)MUL(AT2_ATOMIZE_FLOW,9.663,AT2_ATOMIZE_FLOW_SCFM)MUL(AT3_INLET_FLOW,9.663,AT3_INLET_FLOW_SCFM)MUL(AT3_ATOMIZE_FLOW,9.663,AT3_ATOMIZE_FLOW_SCFM);
END_ROUTINE
